FUNCTION TFDepositoContinuoPalletConsentito : BOOL
VAR_INPUT
	NpacchiPresenti : UINT;
	NpacchiMassimiConsentiti : UINT; // Numero dei pacchi sui trasporti sotto del quale si vuole consentire il deposito continuo dei pallet
	NultimiTrasportiOccupati : uint;
END_VAR
VAR
	i : UINT;
END_VAR

TFDepositoContinuoPalletConsentito := FALSE; 

IF NpacchiPresenti <= NpacchiMassimiConsentiti AND NultimiTrasportiOccupati <= NpacchiMassimiConsentiti THEN
	TFDepositoContinuoPalletConsentito := TRUE;
	RETURN;
ELSE
	TFDepositoContinuoPalletConsentito := FALSE;
	RETURN;
END_IF

END_FUNCTION

(* stored: Version 1.1.0.1, ProductVersion 3.1.4024.11
   POU TFDepositoContinuoPalletConsentito: Id {0f8d1cef-3ff9-45ed-8344-982177652c25}, SpecialFunc None *)
